TYPE CoverTabs :
(
	OVERVIEW := 0,
    TOP := 1,
    BOTTOM := 2,
    IO := 3,
    CONFIG := 4
);
END_TYPE

(* stored: Version 1.1.0.1, ProductVersion 3.1.4018.2
   DUT CoverTabs: Id {0245fdc1-6d9e-47b2-bb87-63ac30ac4444} *)
